// TIA Portal V21 export
DATA_BLOCK "PidParameters"   // DB58
{ S7_Optimized_Access := 'FALSE' }
   VAR RETAIN
      Fv1_Cv01 : Struct
         "Set Value" : Real;
         P : Real := 8.0;
         I : Real := 80.0;
         D : Real := 0.0;
         Mode : Int;
         Output : Real;
         OutputCoil : Bool;
         State : Int;
         Error : Word;
         Reset : Bool;
         InputValue : Real;
      END_STRUCT;
   END_VAR
BEGIN
END_DATA_BLOCK
